FUNCTION_BLOCK FB_MoveVelocity
VAR_INPUT
    Velocity  	: LREAL;
    bExecute   	: BOOL;
    iDirection 	: INT;  // 1 Moving Forward, -1 Moving Backwards
END_VAR

VAR_OUTPUT
    bDone  : BOOL;
    bError : BOOL;
END_VAR

VAR_IN_OUT
	Axis      : AXIS_REF;
END_VAR

VAR
    fbMoveVel : MC_MoveVelocity;
END_VAR

// Move the motor by velocity
fbMoveVel(
    Axis      := Axis,
    Velocity  := Velocity * iDirection,
    Execute   := bExecute
);

bDone := fbMoveVel.InVelocity;
bError := fbMoveVel.Error;

END_FUNCTION_BLOCK

(* stored: Version 1.1.0.1, ProductVersion 3.1.4024.12
   POU FB_MoveVelocity: Id {7db658b2-80b8-4a5a-accc-99a6641d619e}, SpecialFunc None *)
